// TIA Portal V16 export
// export: Created 2022-02-11T10:05:44.5384129Z, ExportSetting WithDefaults, DisplayName Totally Integrated Automation Portal, DisplayVersion V16 Update 5, DisplayName TIA Portal Version Control Interface, DisplayVersion V16 Update 2, DisplayName TIA Portal Openness, DisplayVersion V16 Update 5, DisplayName STEP 7 Professional, DisplayVersion V16 Update 5, DisplayName STEP 7 Safety, DisplayVersion V16, DisplayName WinCC Professional, DisplayVersion V16 Update 5, DisplayName SIMATIC Visualization Architect, DisplayVersion V16
FUNCTION_BLOCK "fbObjMotor_Arrencador"   // FB9211, LAD
{ S7_Optimized_Access := 'TRUE' }
VERSION : 0.1
// stored: AutoNumber false, IsIECCheckEnabled false, IsRetainMemResEnabled true, MemoryReserve 100, RetainMemoryReserve 50, SetENOAutomatically false, UDAEnableTagReadback false
   VAR_INPUT
      aMarxaAuto : Bool := FALSE;   // Activar element mode automatic
      eErrorArrencador : Bool;   // Entrada error proteccio motor filtre
      eReadyArrencador : Bool;
      eConfirmacioMarxa : Bool;   // Senyal confirmacio marxa filtre
      bCM_Marxa : Bool := TRUE;   // Condicions necesaries activar element
      tRegimSoplant : Time := t#30s;
      tAla_ConMar : Time := t#3s;   // Temps retard activacio alarma confirmacio marxa
      tAla_CM : Time := t#2s;   // Temps retard activacio alarma condicions moviment
      tWaitRearranc : Time := T#10s;   // Temps retard entre parada i nova arrencada
      tWaitParada : Time := t#60s;   // Temps espera abans de parada de soplant
      psHabilitada : Bool;
      psEnaAuto : Bool := TRUE;
      psEnaManual : Bool := FALSE;
      psAnuConMov : Bool;
      psResetAlarma : Bool;
      mFirstScan : Bool;
      mPolsosRegim : Bool;
      bSysOk : Bool;
   END_VAR
   VAR_OUTPUT
      aMarxa : Bool;   // Sortida activacio Filtre
      aMarxaNoTimer : Bool;
      be_Marxa : Bool;   // Bit estat Marxa (Confirmacio + Proteccio + Sortida)
      be_Parat : Bool;
      be_Regim : Bool;   // Temps seguretat bomba en marxa
      al_ErrorArrencador : Bool;   // Alarma proteccio motor
      al_NotReady : Bool;
      al_CM : Bool;   // Alarma condicions moviment obrir
      al_Marxa : Bool;   // Alarma confirmacio marxa filtre
      iStatusDisplay : Int;   // Estat visualitzacio EV: 0: Parat, 1; Marxa, 10:Error, 11:Warning
      bDisplayError : Bool;   // Error en EV
      bDisplayWarning : Bool;   // Warning en EV
      bDisplayOk : Bool;   // EV OK
   END_VAR
   VAR
      psManMarxa : Bool;
      be_Marxa_Err : Bool;   // Error en validacio Confirmacio Marxa. Sense retard per alarma.
      bErrorCM : Bool;   // Error CM. Si activem sortida i no es compleixen les CM. Sense retard
      timAla_CM { S7_SetPoint := 'True'} : IEC_TIMER;   // Timer retard alarma condicions moviment
      timAla_Marxa { S7_SetPoint := 'True'} : IEC_TIMER;   // Timer retard alarma marxa filtre
      timDelay_Rearranc { S7_SetPoint := 'True'} : IEC_TIMER;   // Timer retard entre parada i arrencada
      timDelay_Regim { S7_SetPoint := 'True'} : IEC_TIMER;
      timDelay_Parada { S7_SetPoint := 'True'} : IEC_TIMER;
      bCM_Ok { S7_SetPoint := 'True'} : Bool;
      aMarxaSenseTestCM : Bool;   // Bit activacio sortida sense tenir en compte condicions moviment
      bLockWaitStopped : Bool;   // Bloqueig per temps desde ultima parada
      memFlancParo : Bool;
      mAuxTimer : Bool;   // Bit auxiliarInicialitzacio timers
   END_VAR
   VAR_TEMP
      bTmpMarxaAuto : Bool;
      bTmpMarxaMan : Bool;
   END_VAR
   VAR CONSTANT
      STATUS_OBJ_ERR : Int := 10;
      STATUS_OBJ_WARNING : Int := 11;
      STATUS_OBJ_ON : Int := 1;
      STATUS_OBJ_OFF : Int := 0;
      STATUS_OBJ_UNKNOWN : Int := -1;
   END_VAR
   VAR_TEMP   // added for the SCL form of the ladder/FBD networks
      _w1 : Bool;
   END_VAR
BEGIN

REGION Network 1 (SCL)
   // Motor activat per Rele, amb confirmacio i proteccio.
END_REGION

REGION Network 2
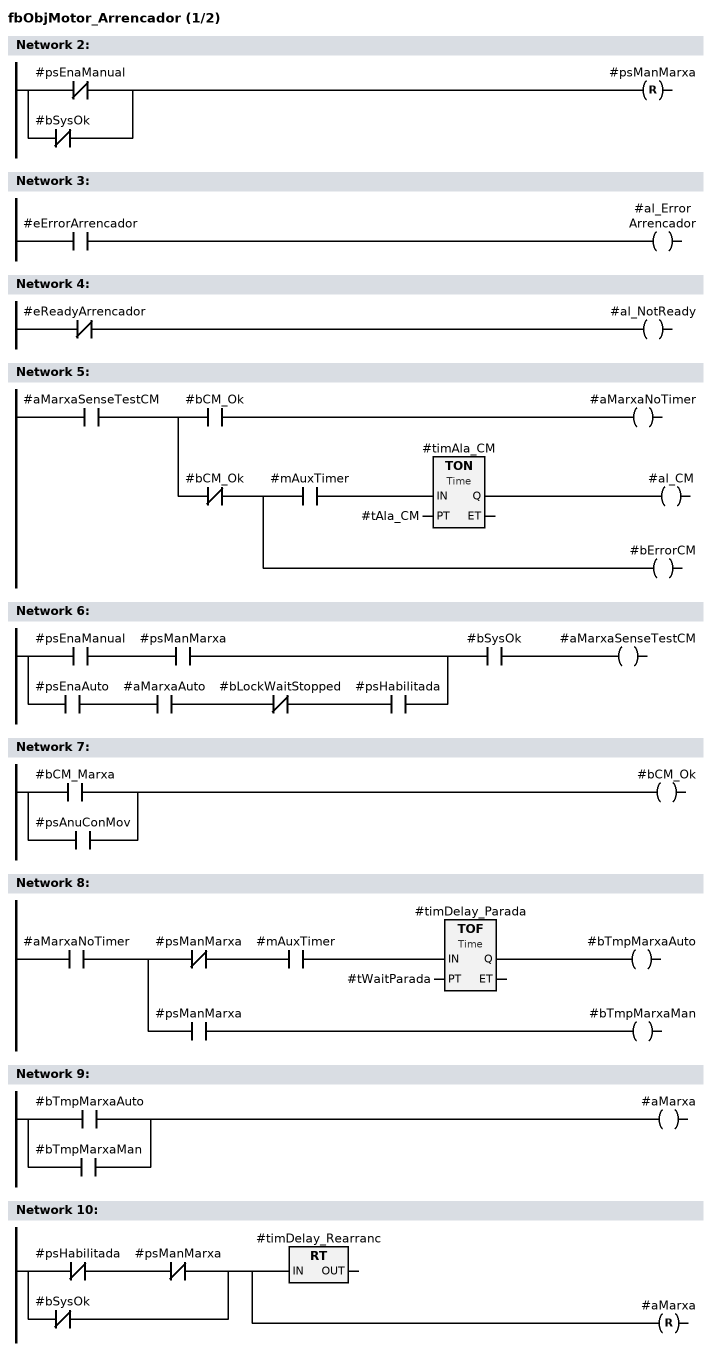
   RUNG wire#powerrail
      I_Contact( #psEnaManual )
      wire#w1
      R_Coil( #psManMarxa )
   END_RUNG
   RUNG wire#powerrail
      I_Contact( #bSysOk )
   END_RUNG wire#w1
   // the same network as SCL:
   IF NOT #psEnaManual OR NOT #bSysOk THEN #psManMarxa := FALSE; END_IF;
END_REGION

REGION Network 3
   RUNG wire#powerrail
      Contact( #eErrorArrencador )
      Coil( #al_ErrorArrencador )
   END_RUNG
   // the same network as SCL:
   #al_ErrorArrencador := #eErrorArrencador;
END_REGION

REGION Network 4
   RUNG wire#powerrail
      I_Contact( #eReadyArrencador )
      Coil( #al_NotReady )
   END_RUNG
   // the same network as SCL:
   #al_NotReady := NOT #eReadyArrencador;
END_REGION

REGION Network 5
   RUNG wire#powerrail
      Contact( #aMarxaSenseTestCM )
      wire#w1
      Contact( #bCM_Ok )
      Coil( #aMarxaNoTimer )
   END_RUNG
   RUNG wire#w1
      I_Contact( #bCM_Ok )
      wire#w2
      Contact( #mAuxTimer )
      { S7_Templates := "time_type := Time" } #timAla_CM.TON(pt := #tAla_CM, et =>)
      Coil( #al_CM )
   END_RUNG
   RUNG wire#w2
      Coil( #bErrorCM )
   END_RUNG
   // the same network as SCL:
   #aMarxaNoTimer := #aMarxaSenseTestCM AND #bCM_Ok;
   #_w1 := #aMarxaSenseTestCM AND NOT #bCM_Ok;
   #timAla_CM.TON(IN := #_w1 AND #mAuxTimer, PT := #tAla_CM);
   #al_CM := #timAla_CM.Q;
   #bErrorCM := #_w1;
END_REGION

REGION Network 6
   RUNG wire#powerrail
      Contact( #psEnaManual )
      Contact( #psManMarxa )
      wire#w1
      Contact( #bSysOk )
      Coil( #aMarxaSenseTestCM )
   END_RUNG
   RUNG wire#powerrail
      Contact( #psEnaAuto )
      Contact( #aMarxaAuto )
      I_Contact( #bLockWaitStopped )
      Contact( #psHabilitada )
   END_RUNG wire#w1
   // the same network as SCL:
   #aMarxaSenseTestCM := ((#psEnaManual AND #psManMarxa) OR (#psEnaAuto AND #aMarxaAuto AND NOT #bLockWaitStopped AND #psHabilitada)) AND #bSysOk;
END_REGION

REGION Network 7
   RUNG wire#powerrail
      Contact( #bCM_Marxa )
      wire#w1
      Coil( #bCM_Ok )
   END_RUNG
   RUNG wire#powerrail
      Contact( #psAnuConMov )
   END_RUNG wire#w1
   // the same network as SCL:
   #bCM_Ok := #bCM_Marxa OR #psAnuConMov;
END_REGION

REGION Network 8
   RUNG wire#powerrail
      Contact( #aMarxaNoTimer )
      wire#w1
      I_Contact( #psManMarxa )
      Contact( #mAuxTimer )
      { S7_Templates := "time_type := Time" } #timDelay_Parada.TOF(pt := #tWaitParada, et =>)
      Coil( #bTmpMarxaAuto )
   END_RUNG
   RUNG wire#w1
      Contact( #psManMarxa )
      Coil( #bTmpMarxaMan )
   END_RUNG
   // the same network as SCL:
   #timDelay_Parada.TOF(IN := #aMarxaNoTimer AND NOT #psManMarxa AND #mAuxTimer, PT := #tWaitParada);
   #bTmpMarxaAuto := #timDelay_Parada.Q;
   #bTmpMarxaMan := #aMarxaNoTimer AND #psManMarxa;
END_REGION

REGION Network 9
   RUNG wire#powerrail
      Contact( #bTmpMarxaAuto )
      wire#w1
      Coil( #aMarxa )
   END_RUNG
   RUNG wire#powerrail
      Contact( #bTmpMarxaMan )
   END_RUNG wire#w1
   // the same network as SCL:
   #aMarxa := #bTmpMarxaAuto OR #bTmpMarxaMan;
END_REGION

REGION Network 10
   RUNG wire#powerrail
      I_Contact( #psHabilitada )
      I_Contact( #psManMarxa )
      wire#w1
      RT_Coil( #timDelay_Rearranc )
   END_RUNG
   RUNG wire#powerrail
      I_Contact( #bSysOk )
   END_RUNG wire#w1
   RUNG wire#w1
      R_Coil( #aMarxa )
   END_RUNG
   // the same network as SCL:
   #_w1 := (NOT #psHabilitada AND NOT #psManMarxa) OR NOT #bSysOk;
   IF #_w1 THEN
       RESET_TIMER(#timDelay_Rearranc);
       #aMarxa := FALSE;
   END_IF;
END_REGION

REGION Network 11
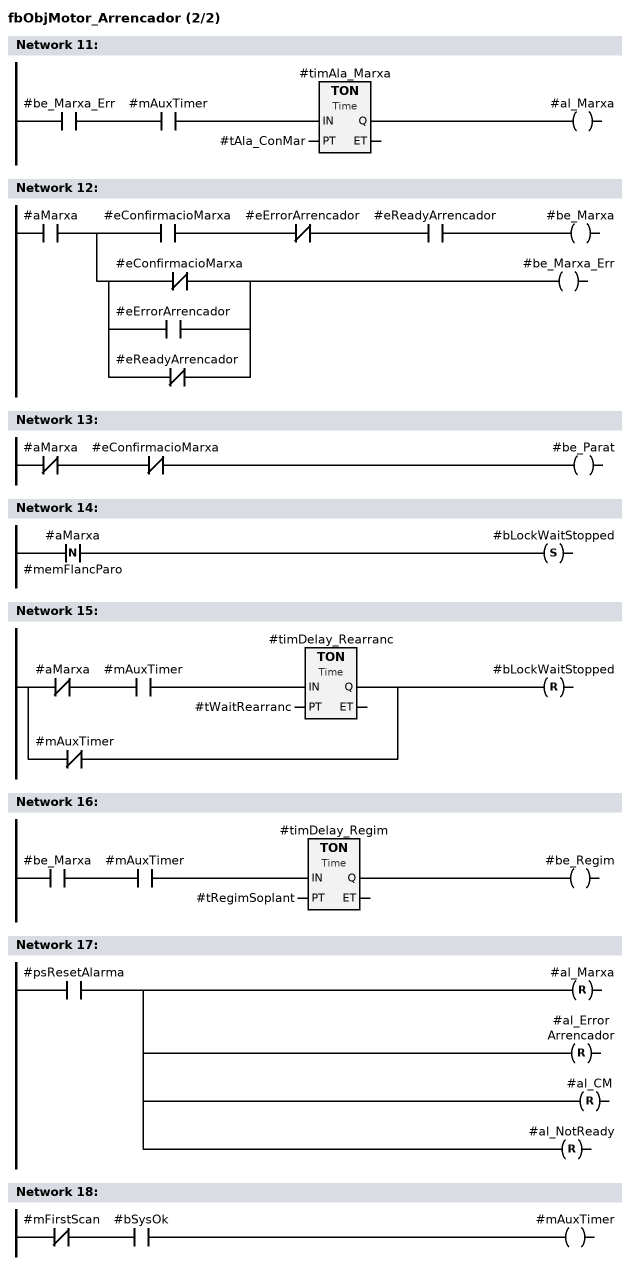
   RUNG wire#powerrail
      Contact( #be_Marxa_Err )
      Contact( #mAuxTimer )
      { S7_Templates := "time_type := Time" } #timAla_Marxa.TON(pt := #tAla_ConMar, et =>)
      Coil( #al_Marxa )
   END_RUNG
   // the same network as SCL:
   #timAla_Marxa.TON(IN := #be_Marxa_Err AND #mAuxTimer, PT := #tAla_ConMar);
   #al_Marxa := #timAla_Marxa.Q;
END_REGION

REGION Network 12
   RUNG wire#powerrail
      Contact( #aMarxa )
      wire#w1
      Contact( #eConfirmacioMarxa )
      I_Contact( #eErrorArrencador )
      Contact( #eReadyArrencador )
      Coil( #be_Marxa )
   END_RUNG
   RUNG wire#w1
      I_Contact( #eConfirmacioMarxa )
      wire#w2
      Coil( #be_Marxa_Err )
   END_RUNG
   RUNG wire#w1
      Contact( #eErrorArrencador )
   END_RUNG wire#w2
   RUNG wire#w1
      I_Contact( #eReadyArrencador )
   END_RUNG wire#w2
   // the same network as SCL:
   #be_Marxa := #aMarxa AND #eConfirmacioMarxa AND NOT #eErrorArrencador AND #eReadyArrencador;
   #be_Marxa_Err := #aMarxa AND (NOT #eConfirmacioMarxa OR #eErrorArrencador OR NOT #eReadyArrencador);
END_REGION

REGION Network 13
   RUNG wire#powerrail
      I_Contact( #aMarxa )
      I_Contact( #eConfirmacioMarxa )
      Coil( #be_Parat )
   END_RUNG
   // the same network as SCL:
   #be_Parat := NOT #aMarxa AND NOT #eConfirmacioMarxa;
END_REGION

REGION Network 14
   RUNG wire#powerrail
      N_Contact(operand := #aMarxa, bit := #memFlancParo)
      S_Coil( #bLockWaitStopped )
   END_RUNG
   // the same network as SCL:
   #_w1 := NOT #aMarxa AND #memFlancParo;   // falling edge of #aMarxa
   #memFlancParo := #aMarxa;
   IF #_w1 THEN #bLockWaitStopped := TRUE; END_IF;
END_REGION

REGION Network 15
   RUNG wire#powerrail
      I_Contact( #aMarxa )
      Contact( #mAuxTimer )
      { S7_Templates := "time_type := Time" } #timDelay_Rearranc.TON(pt := #tWaitRearranc, et =>)
      wire#w1
      R_Coil( #bLockWaitStopped )
   END_RUNG
   RUNG wire#powerrail
      I_Contact( #mAuxTimer )
   END_RUNG wire#w1
   // the same network as SCL:
   #timDelay_Rearranc.TON(IN := NOT #aMarxa AND #mAuxTimer, PT := #tWaitRearranc);
   IF #timDelay_Rearranc.Q OR NOT #mAuxTimer THEN #bLockWaitStopped := FALSE; END_IF;
END_REGION

REGION Network 16
   RUNG wire#powerrail
      Contact( #be_Marxa )
      Contact( #mAuxTimer )
      { S7_Templates := "time_type := Time" } #timDelay_Regim.TON(pt := #tRegimSoplant, et =>)
      Coil( #be_Regim )
   END_RUNG
   // the same network as SCL:
   #timDelay_Regim.TON(IN := #be_Marxa AND #mAuxTimer, PT := #tRegimSoplant);
   #be_Regim := #timDelay_Regim.Q;
END_REGION

REGION Network 17
   RUNG wire#powerrail
      Contact( #psResetAlarma )
      wire#w1
      R_Coil( #al_Marxa )
   END_RUNG
   RUNG wire#w1
      R_Coil( #al_ErrorArrencador )
   END_RUNG
   RUNG wire#w1
      R_Coil( #al_CM )
   END_RUNG
   RUNG wire#w1
      R_Coil( #al_NotReady )
   END_RUNG
   // the same network as SCL:
   IF #psResetAlarma THEN
       #al_Marxa := FALSE;
       #al_ErrorArrencador := FALSE;
       #al_CM := FALSE;
       #al_NotReady := FALSE;
   END_IF;
END_REGION

REGION Network 18
   RUNG wire#powerrail
      I_Contact( #mFirstScan )
      Contact( #bSysOk )
      Coil( #mAuxTimer )
   END_RUNG
   // the same network as SCL:
   #mAuxTimer := NOT #mFirstScan AND #bSysOk;
END_REGION

REGION Network 19 (SCL)
       IF (#al_Marxa OR #al_CM OR #al_ErrorArrencador OR #al_NotReady) THEN
           #iStatusDisplay := #STATUS_OBJ_ERR;                // Error = 10
           #bDisplayError := TRUE;
           #bDisplayWarning := FALSE;
           #bDisplayOk := FALSE;

       ELSIF (#be_Marxa_Err OR #bErrorCM) OR #bLockWaitStopped THEN
           #iStatusDisplay := #STATUS_OBJ_WARNING;            // Warning = 11
           #bDisplayError := FALSE;
           #bDisplayWarning := TRUE;
           #bDisplayOk := FALSE;

       ELSIF ((#aMarxa) AND (NOT #aMarxaNoTimer)) THEN    // Temps seguretat marxa     
           IF #mPolsosRegim THEN
               #iStatusDisplay := #STATUS_OBJ_ON;                 // Bit estat Marxa Auto = 1
           ELSE
               #iStatusDisplay := #STATUS_OBJ_OFF;
           END_IF;
           #bDisplayError := FALSE;
           #bDisplayWarning := FALSE;
           #bDisplayOk := TRUE;

       ELSIF #be_Regim THEN
           #iStatusDisplay := #STATUS_OBJ_ON;                 // Bit estat Marxa Auto = 1
           #bDisplayError := FALSE;
           #bDisplayWarning := FALSE;
           #bDisplayOk := TRUE;

       ELSIF #be_Marxa THEN
           IF #mPolsosRegim THEN
               #iStatusDisplay := #STATUS_OBJ_ON;                 // Bit estat Marxa Auto = 1
           ELSE
               #iStatusDisplay := #STATUS_OBJ_WARNING;
           END_IF;
           #bDisplayError := FALSE;
           #bDisplayWarning := FALSE;
           #bDisplayOk := TRUE;

       ELSIF #aMarxa THEN
           #iStatusDisplay := #STATUS_OBJ_WARNING;            // Bit estat Arrancant = 6
           #bDisplayError := FALSE;
           #bDisplayWarning := TRUE;
           #bDisplayOk := FALSE;

       ELSE
           #iStatusDisplay := #STATUS_OBJ_OFF;                // Bit estat Stop
           #bDisplayError := FALSE;
           #bDisplayWarning := FALSE;
           #bDisplayOk := TRUE;

       END_IF;
END_REGION
END_FUNCTION_BLOCK
